FUNCTION_BLOCK FB_MasterArm
VAR
	// arm index, 1 for left arm, 2 for right arm
	m_armIdx: INT;
	
	// grip angle calculator
	m_gripHallSensorIO AT%I* :UDINT;	
	m_gripAngleCalc : FB_GripAngleCalc;
	m_gripAngle :LREAL;
	
	//hand clutch switch IO
	m_handClutchIO AT%I*:UDINT;
	m_handClutchCheck :FB_HandClutchCheck;
	m_handClutchSwitch :BOOL;
	
	// joints
	// NOTICE: all joints are the true active joints, not DH ones!
	m_joints :ARRAY[1..g_mJntNum] OF FB_ArmJoint;
	
	// master gripper roll flip flag, if true, q7 would add pi in FK
	m_gripperRollFlip :BOOL :=False;
	
	// arm cartesian data, defined in each arm origin
	m_curCartPose	:ST_Frame;
	m_curCartTwist: Vec6d;
	m_cmdCartTwist :Vec6d;
	m_cmdCartPose:ST_Frame;
	m_curCartLinkPose :ST_Frame;
	m_curCartLinkTwist :Vec6d;
	
	
	// arm joint data
	m_curMotorPos :Vec7d;
	m_curLinkPos :Vec7d;
	m_curJntPos :Vec7d;
	m_curJntVel :Vec7d;
	m_curLinkVel :Vec7d;
	m_curJntTrq :Vec7d;
	m_rawJntCurrent :Vec7d;
	m_filtJntCurrent :Vec7d;
	m_cmdJntCurrent : Vec7d;
	m_cmdJntTrq :Vec7d;
	m_cmdJntPos :Vec7d;
	m_cmdJntVel :Vec7d;

	
	// arm dynamic data
	m_jntGravity : Vec7d;
	m_jntMassMat : Mat7d;
	m_lambda :Mat6d;
	m_dynaNullspace :Mat7d;
	m_jntFriction :Vec7d;
	m_jntExtTrq :Vec7d;
	
	// arm jacobian 
	m_jaco : Mat67;
	m_linkJaco : Mat67;
	
	// simulated status
	m_simJntPos :Vec7d;
	m_simCartPose : ST_Frame;
	m_simJaco : Mat67;
	
	// joint position controller
	m_jntPIDCtrl :ARRAY[1..g_mJntNum] OF FB_PID;
	
	//inertia compensation---1106
	m_curJntAcc :Vec7d;
	m_curLinkAcc :Vec7d;
	m_jntInertiaTrq:Vec7d;
	m_linkInertiaTrq:Vec7d;	
	
	//Calculate space velocity related variables
	m_linkJacoLast : Mat67; //last link jacobian matrix
	m_spaceAcc:Vec6d; //space acceleration
	m_spaceAccByDiff:Vec6d;
	m_curCartLinkTwistLast :Vec6d;	
	
	//Spatial force related variables
	m_spatialForce:Vec6d;
	m_spatialForceByAccDiff:Vec6d;
	m_jntTorForAcc:Vec7d;
	m_jntTorForAccByDiff:Vec7d;
	
	//Spatial acceleration filter
	m_spatialAccLpf :ARRAY[1..6] OF FB_LowPassFilter;
	m_spatialAccLpf_2 :ARRAY[1..6] OF FB_LowPassFilter;
END_VAR

PROPERTY armIdx : int
GET
armIdx:=m_armIdx;
END_GET
END_PROPERTY

METHOD PROTECTED calcJaco : BOOL
VAR_IN_OUT CONSTANT
	i_jntPos :ARRAY[1..g_mJntNum] OF LREAL;
END_VAR
VAR_IN_OUT
	r_jaco :ARRAY[1..g_cartDofs, 1..g_mJntNum] OF LREAL;
END_VAR
VAR_INPUT
END_VAR

VAR
	q1,q2, q3, q4, q5, q6, q7 :LREAL;
	d1,d4,a3,a4 :LREAL;
	c1,c2,c3,c4,c5,c6,c7 :LREAL;
	s1,s2,s3,s4,s5,s6,s7 :LREAL;
	c23, s23 :LREAL;
	j:INT;
END_VAR
// !Convert active joint position to DH model for kinematic calculation
q1:=i_jntPos[1];  
q2:=i_jntPos[2];  
q3:=i_jntPos[3]-i_jntPos[2];  //q3=q8-q2
q4:=i_jntPos[4]+i_jntPos[3]-i_jntPos[2]-pi/2;//q4DH=q4motor+q8-q2-90;  
q5:=i_jntPos[5];  
q6:=i_jntPos[6];  
q7:=i_jntPos[7];  
d1:=g_d1;
d4:=g_d4;
a3:=g_a3;
a4:=g_a4;
c1:=COS(q1);
c2:=COS(q2);
c3:=COS(q3);
c4:=COS(q4);
c5:=COS(q5);
c6:=COS(q6);
c7:=COS(q7);
s1:=SIN(q1);
s2:=SIN(q2);
s3:=SIN(q3);
s4:=SIN(q4);
s5:=SIN(q5);
s6:=SIN(q6);
s7:=SIN(q7);
c23:=COS(q2+q3);
s23:=SIN(q2+q3);

// jacobian with DH joints
r_jaco[1,1]:=-s1*(c2*(a3 + a4*c3 - d4*s3) - s2*(d4*c3 + a4*s3)) ;
r_jaco[1,2]:=-c1*(s2*(a3 + a4*c3 - d4*s3) + c2*(d4*c3 + a4*s3)) ;
r_jaco[1,3]:=-c1*(d4*c23 + a4*s23) ;
r_jaco[1,4]:=0 ;
r_jaco[1,5]:=0 ;
r_jaco[1,6]:=0 ;
r_jaco[1,7]:=0;
 
r_jaco[2,1]:=c1*(c2*(a3 + a4*c3 - d4*s3) - s2*(d4*c3 + a4*s3)); 
r_jaco[2,2]:=-s1*(s2*(a3 + a4*c3 - d4*s3) + c2*(d4*c3 + a4*s3)); 
r_jaco[2,3]:=-s1*(d4*c23 + a4*s23); 
r_jaco[2,4]:=0; 
r_jaco[2,5]:=0; 
r_jaco[2,6]:=0; 
r_jaco[2,7]:=0;

 
r_jaco[3,1]:=0 ;
r_jaco[3,2]:=- c1*(c1*c2*(a3 + a4*c3 - d4*s3) - c1*s2*(d4*c3 + a4*s3)) - s1*(c2*s1*(a3 + a4*c3 - d4*s3) - s1*s2*(d4*c3 + a4*s3));
r_jaco[3,3]:=- c1*(a4*c23*c1 - d4*s23*c1) - s1*(a4*c23*s1 - d4*s23*s1);
r_jaco[3,4]:=0;
r_jaco[3,5]:=0;
r_jaco[3,6]:=0 ;
r_jaco[3,7]:=0 ;

r_jaco[4,1]:=0 ;
r_jaco[4,2]:=-s1 ;
r_jaco[4,3]:=-s1 ;
r_jaco[4,4]:=-s23*c1 ;
r_jaco[4,5]:=c23*c1*s4 - c4*s1 ;
r_jaco[4,6]:=- s5*(s1*s4 + c23*c1*c4) - s23*c1*c5 ;
r_jaco[4,7]:=s6*(c5*(s1*s4 + c4*(c1*c2*c3 - c1*s2*s3)) - s5*(c1*c2*s3 + c1*c3*s2)) - c6*(c4*s1 - s4*(c1*c2*c3 - c1*s2*s3));
 
r_jaco[5,1]:=0; 
r_jaco[5,2]:=c1; 
r_jaco[5,3]:=c1; 
r_jaco[5,4]:=-s23*s1; 
r_jaco[5,5]:=c1*c4 + c23*s1*s4; 
r_jaco[5,6]:=s5*(c1*s4 - c23*c4*s1) - s23*c5*s1; 
r_jaco[5,7]:=c6*(c1*c4 - s4*(s1*s2*s3 - c2*c3*s1)) - s6*(c5*(c1*s4 + c4*(s1*s2*s3 - c2*c3*s1)) + s5*(c2*s1*s3 + c3*s1*s2));

r_jaco[6,1]:=1 ;
r_jaco[6,2]:=0 ;
r_jaco[6,3]:=0 ;
r_jaco[6,4]:=-c23 ;
r_jaco[6,5]:=-s23*s4 ;
r_jaco[6,6]:=s23*c4*s5 - c23*c5 ;
r_jaco[6,7]:=- s6*(c23*s5 + s23*c4*c5) - s23*c6*s4;

// jacobian with active joints
// jaco_DH*qdot_DH = jaco_DH * (A * qdot)= jaco * qdot
// A =[ 1  0 0 0 0 0 0
//		0  1 0 0 0 0 0
//		0 -1 1 0 0 0 0
//		0 -1 1 1 0 0 0
//		0 0  0 0 1 0 0
//      0 0  0 0 0 1 0
// 		0 0  0 0 0 0 1]
 FOR j:=1 TO 6 DO 
	 r_jaco[j,2]:=r_jaco[j,2]-r_jaco[j,3]-r_jaco[j,4];
	 r_jaco[j,3]:=r_jaco[j,3]+r_jaco[j,4];
 END_FOR
END_METHOD

PROPERTY cmdCartPose : REFERENCE TO ST_Frame
GET
cmdCartPose REF= m_cmdCartPose;
END_GET
END_PROPERTY

PROPERTY cmdCartTwist : REFERENCE to Vec6d
GET
cmdCartTwist REF= m_cmdCartTwist;
END_GET
END_PROPERTY

PROPERTY cmdJntCurrent :REFERENCE to Vec7d
GET
cmdJntCurrent REF= m_cmdJntCurrent;
END_GET
END_PROPERTY

PROPERTY cmdJntPos : REFERENCE TO Vec7d
GET
cmdJntPos REF= m_cmdJntPos;
END_GET
END_PROPERTY

PROPERTY cmdJntTrq :REFERENCE TO Vec7d
GET
cmdJntTrq REF= m_cmdJntTrq;
END_GET
END_PROPERTY

PROPERTY cmdJntVel : REFERENCE TO Vec7d
GET
cmdJntVel REF= m_cmdJntVel;
END_GET
END_PROPERTY

PROPERTY curCartPose :REFERENCE to ST_Frame
GET
curCartPose REF=m_curCartPose;
END_GET
END_PROPERTY

PROPERTY curCartTwist :REFERENCE TO Vec6d
GET
curCartTwist REF=m_curCartTwist;
END_GET
END_PROPERTY

PROPERTY curJntInertiaTrq :REFERENCE TO Vec7d
GET

//cmdJntPos REF= m_cmdJntPos;---inertia compensation---1106
IF (gvl.m_InertiaSelect[m_armIdx]=1) THEN
	curJntInertiaTrq REF=m_jntInertiaTrq;
	
ELSIF(gvl.m_InertiaSelect[m_armIdx]=2) THEN
	curJntInertiaTrq REF=m_linkInertiaTrq;
	
ELSIF(gvl.m_InertiaSelect[m_armIdx]=3) THEN
	curJntInertiaTrq REF=m_jntTorForAcc;
	
ELSIF(gvl.m_InertiaSelect[m_armIdx]=4) THEN
	curJntInertiaTrq REF=m_jntTorForAccByDiff;
END_IF
END_GET
SET
END_SET
END_PROPERTY

PROPERTY curJntPos :REFERENCE TO Vec7d
GET
curJntPos REF=m_curJntPos;
END_GET
END_PROPERTY

PROPERTY curJntTrq :REFERENCE TO Vec7d
GET
curJntTrq REF=m_curJntTrq;
END_GET
END_PROPERTY

PROPERTY curJntVel :REFERENCE TO Vec7d
GET
curJntVel REF=m_curJntVel;
END_GET
END_PROPERTY

PROPERTY curLinkPos :REFERENCE TO  Vec7d
GET
curLinkPos REF=m_curLinkPos;
END_GET
END_PROPERTY

PROPERTY curMotorPos :REFERENCE TO Vec7d
GET
curMotorPos REF=m_curMotorPos;
END_GET
END_PROPERTY

PROPERTY PUBLIC dynaNullspace : REFERENCE TO Mat7d
GET
dynaNullspace REF= m_dynaNullspace;
END_GET
END_PROPERTY

METHOD PROTECTED enable : BOOL
VAR_IN_OUT CONSTANT
	i_jntIdx :Vec7i;
END_VAR
VAR
	i :INT ;
END_VAR
FOR i:=1 TO g_mJntNum DO
	IF 1= i_jntIdx[i] THEN
		m_joints[i].enable();
	ELSE
		m_joints[i].disable();
	END_IF
END_FOR
END_METHOD

PROPERTY filtJntCurrent :REFERENCE to Vec7d
GET
filtJntCurrent ref= m_filtJntCurrent;
END_GET
END_PROPERTY

METHOD PUBLIC flipGripper : BOOL
VAR_INPUT
	i_flipFlag :BOOL;
END_VAR
m_gripperRollFlip := i_flipFlag;
END_METHOD

// from active joint position to cartesian pose in arm origin
METHOD PROTECTED forwardKinematic : BOOL
VAR_IN_OUT CONSTANT
	i_jntPos :ARRAY[1..g_mJntNum] OF LREAL;
END_VAR
VAR_IN_OUT
	r_cartPose :ST_Frame;
END_VAR
VAR
	q1,q2, q3, q4, q5, q6, q7 :LREAL;
	d1,d4,a3,a4 :LREAL;
	c1,c2,c3,c4,c5,c6,c7 :LREAL;
	s1,s2,s3,s4,s5,s6,s7 :LREAL;
	c23, s23 :LREAL;
END_VAR
// !Convert active joint position to DH model for kinematic calculation
q1:=i_jntPos[1];  
q2:=i_jntPos[2];  
q3:=i_jntPos[3]-i_jntPos[2];  //q3=q8-q2
q4:=jnt4MotorToLink(i_jntPos[2],i_jntPos[3], i_jntPos[4]);//q4DH=q4motor+q8-q2-90;  
q5:=i_jntPos[5];  
q6:=i_jntPos[6];  
q7:=i_jntPos[7];  

// master roll flip handle
IF m_gripperRollFlip THEN
	q7 := q7+PI;
END_IF

d1:=g_d1;
d4:=g_d4;
a3:=g_a3;
a4:=g_a4;
c1:=COS(q1);
c2:=COS(q2);
c3:=COS(q3);
c4:=COS(q4);
c5:=COS(q5);
c6:=COS(q6);
c7:=COS(q7);
s1:=SIN(q1);
s2:=SIN(q2);
s3:=SIN(q3);
s4:=SIN(q4);
s5:=SIN(q5);
s6:=SIN(q6);
s7:=SIN(q7);
c23:=COS(q2+q3);
s23:=SIN(q2+q3);

// cartesian pose frame
r_cartPose.m_pos[1]:=c1*(a4*c23 - d4*s23 + a3*c2); 
r_cartPose.m_pos[2]:=s1*(a4*c23 - d4*s23 + a3*c2);
r_cartPose.m_pos[3]:=d1 - d4*c23 - a4*s23 - a3*s2;  
r_cartPose.m_rot[1,1]:=c7*(s6*(c4*s1 - s4*(c1*c2*c3 - c1*s2*s3)) + c6*(c5*(s1*s4 + c4*(c1*c2*c3 - c1*s2*s3)) - s5*(c1*c2*s3 + c1*c3*s2))) - s7*(s5*(s1*s4 + c4*(c1*c2*c3 - c1*s2*s3)) + c5*(c1*c2*s3 + c1*c3*s2));
r_cartPose.m_rot[2,1]:=s7*(s5*(c1*s4 + c4*(s1*s2*s3 - c2*c3*s1)) - c5*(c2*s1*s3 + c3*s1*s2)) - c7*(s6*(c1*c4 - s4*(s1*s2*s3 - c2*c3*s1)) + c6*(c5*(c1*s4 + c4*(s1*s2*s3 - c2*c3*s1)) + s5*(c2*s1*s3 + c3*s1*s2)));
r_cartPose.m_rot[3,1]:=- s7*(c23*c5 - s23*c4*s5) - c7*(c23*c6*s5 - s23*s4*s6 + s23*c4*c5*c6); 
r_cartPose.m_rot[1,2]:=- s7*(s6*(c4*s1 - s4*(c1*c2*c3 - c1*s2*s3)) + c6*(c5*(s1*s4 + c4*(c1*c2*c3 - c1*s2*s3)) - s5*(c1*c2*s3 + c1*c3*s2))) - c7*(s5*(s1*s4 + c4*(c1*c2*c3 - c1*s2*s3)) + c5*(c1*c2*s3 + c1*c3*s2)); 
r_cartPose.m_rot[2,2]:=s7*(s6*(c1*c4 - s4*(s1*s2*s3 - c2*c3*s1)) + c6*(c5*(c1*s4 + c4*(s1*s2*s3 - c2*c3*s1)) + s5*(c2*s1*s3 + c3*s1*s2))) + c7*(s5*(c1*s4 + c4*(s1*s2*s3 - c2*c3*s1)) - c5*(c2*s1*s3 + c3*s1*s2)); 
r_cartPose.m_rot[3,2]:=s7*(c23*c6*s5 - s23*s4*s6 + s23*c4*c5*c6) - c7*(c23*c5 - s23*c4*s5); 
r_cartPose.m_rot[1,3]:=s6*(c5*(s1*s4 + c4*(c1*c2*c3 - c1*s2*s3)) - s5*(c1*c2*s3 + c1*c3*s2)) - c6*(c4*s1 - s4*(c1*c2*c3 - c1*s2*s3)); 
r_cartPose.m_rot[2,3]:=c6*(c1*c4 - s4*(s1*s2*s3 - c2*c3*s1)) - s6*(c5*(c1*s4 + c4*(s1*s2*s3 - c2*c3*s1)) + s5*(c2*s1*s3 + c3*s1*s2));
r_cartPose.m_rot[3,3]:=- s6*(c23*s5 + s23*c4*c5) - s23*c6*s4;
END_METHOD

PROPERTY gripAngle : LREAL
GET
gripAngle:=m_gripAngle;
END_GET
END_PROPERTY

PROPERTY gripperRollFlip : BOOL
GET
gripperRollFlip := m_gripperRollFlip;
END_GET
END_PROPERTY

PROPERTY handClutchSwitch : BOOL
GET
handClutchSwitch :=m_handClutchSwitch;
END_GET
END_PROPERTY

METHOD PUBLIC init : BOOL
VAR_INPUT
	i_armIdx:INT;
END_VAR
VAR 
	i :INT ;
	currentRatioMotor2Jnt: LREAL;
END_VAR
// arm statues init
m_armIdx:=i_armIdx;
m_gripAngle:=0;
m_gripAngleCalc.init(m_armIdx);

// joint init
FOR i:=1 TO g_mJntNum DO
	m_joints[i].init(m_armIdx, i,g_armCtrlCycleTime);
END_FOR

// init joint encoder and position calculation
initJntPos();

// joint controller init
FOR i:=1 TO g_mJntNum DO 
	currentRatioMotor2Jnt:=GVL_ArmJointParameters.g_motorTrqConst[i]*GVL_ArmJointParameters.g_motorReduction[i]/1000;
	m_jntPIDCtrl[i].init(g_armCtrlCycleTime,g_posKp[i],g_posKd[i],g_posKi[i],
		g_posKiLimit[i]* currentRatioMotor2Jnt,	g_posCtrlLimit[i]*currentRatioMotor2Jnt);
END_FOR

//spatial acceleration init---inertia compensation---1106
FOR i:=1 TO 6 DO 
	m_spatialAccLpf[i].init(1, g_curJntVelLpfCutoffFreq*0.2, g_armCtrlFreq/gvl.g_accCalCycle);
	m_spatialAccLpf_2[i].init(1, g_curJntVelLpfCutoffFreq*0.2, g_armCtrlFreq/gvl.g_accCalCycle);
END_FOR
END_METHOD

METHOD public initJntPos : BOOL
VAR_INPUT
END_VAR
VAR
	i:INT ;
	initLinkPos:LREAL;
END_VAR
// joint init
FOR i:=1 TO g_mJntNum DO
	m_joints[i].initJntPos();
END_FOR

// link position of joint4 is influenced by joint2 and joint3, need to handle seperately
initLinkPos:=jnt4LinkToMotor(m_joints[2].initLinkPos,m_joints[3].initLinkPos, m_joints[4].initLinkPos);
m_joints[4].initJntPosReset(initLinkPos);

// update arm status after joint position is re-init
updateStatus();
END_METHOD

// from cartesian pose in arm origin to active joint position
METHOD PROTECTED inverseKinematic : BOOL
VAR_INPUT
	q4:LREAL;
	solution_ID:INT;
END_VAR
VAR_IN_OUT CONSTANT
	i_curCartPose :ST_Frame;
END_VAR
VAR_IN_OUT
	r_jntPos :ARRAY[1..g_mJntNum] OF LREAL;
END_VAR
VAR
	a3,a4,d1,d4:LREAL;
	px,py,pz:lreal;
	nx,ny,nz:lreal;
	ox,oy,oz:lreal;
	ax,ay,az:lreal;

	q1,q2,q3,q5,q6,q7:LREAL;
	
	q11,q12:LREAL;
	k1,A,B,C,fi,R0,q21,q22:lreal;
	ins1,ins2:lreal;
	
	A11,A12,A21,A22,C1,C2:lreal;
	SIN23,COS23,q23:lreal;
	
	T_74_left_23,q61,q62:lreal;
	T_74_left_13,T_74_left_33:lreal;
	T_74_left_21,T_74_left_22:LREAL;	
	
	succeed_1,succeed_2,succeed:BOOL;
END_VAR


//***********************单臂逆向运动学**************************//
d1:=g_d1;
d4:=g_d4;
a3:=g_a3;
a4:=g_a4;

nx:=i_curCartPose.m_rot[1,1];  ny:=i_curCartPose.m_rot[2,1];  nz:=i_curCartPose.m_rot[3,1];
ox:=i_curCartPose.m_rot[1,2]; oy:=i_curCartPose.m_rot[2,2];  oz:=i_curCartPose.m_rot[3,2];
ax:=i_curCartPose.m_rot[1,3];  ay:=i_curCartPose.m_rot[2,3];  az:=i_curCartPose.m_rot[3,3];
px:=i_curCartPose.m_pos[1]; py:=i_curCartPose.m_pos[2]; pz:=i_curCartPose.m_pos[3];


//求解q1
q11:=atan2(y:= py, x:= px);
q12:=-q11;
IF (Solution_ID<=4) THEN
	q1:=q11;
ELSE
	q1:=q12;
END_IF



//求解q2
k1:=px*COS(q1) + py*SIN(q1);
A:=2*a3*pz - 2*a3*d1;
B:=2*a3*k1;
C:=a3*a3 - a4*a4 + d1*d1 - 2*d1*pz - d4*d4 + k1*k1 + pz*pz;
fi:=atan2(y:= B, x:= A);

R0:=SQRT(A*A+B*B);

//*************程序保护性处理，避免软件崩溃***************//
IF ABS(C/R0)>1 THEN
	succeed_1:=FALSE;
	succeed:=FALSE;
	RETURN;
ELSE
	succeed_1:=TRUE;
END_IF

ins1:=atan2(y:= C/R0, x:= SQRT(1-(C/R0)*(C/R0)));
q21:=fi-ins1;
ins2:=atan2(y:= C/R0, x:= -SQRT(1-(C/R0)*(C/R0)));
q22:=fi-ins2;

IF (Solution_ID=1) OR (Solution_ID=2) OR (Solution_ID=5) OR (Solution_ID=6) THEN
	q2:=q21;
ELSE
	q2:=q22;
END_IF




//求解q3
A11:=- d4;
A12:=a4;
A21:=- a4;
A22:=-d4;
C1:=k1- a3*COS(q2);
C2:=pz - d1 + a3*SIN(q2);
sin23:=(C1*A22-C2*A12)/(A11*A22-A21*A12);
cos23:=(C2*A11-C1*A21)/(A11*A22-A21*A12);
q23:=atan2(y:= sin23, x:= cos23);
q3:=q23-q2;




//求解q6
T_74_left_23:=ax*(COS(q4)*SIN(q1) - COS(q1)*COS(q2)*COS(q3)*SIN(q4) + COS(q1)*SIN(q2)*SIN(q3)*SIN(q4)) - ay*(COS(q1)*COS(q4) + COS(q2)*COS(q3)*SIN(q1)*SIN(q4) - SIN(q1)*SIN(q2)*SIN(q3)*SIN(q4)) + az*SIN(q2 + q3)*SIN(q4);

//*************程序保护性处理，避免软件崩溃***************//
IF ABS(T_74_left_23>1) THEN
	succeed_2:=FALSE;
	succeed:=FALSE;
	RETURN;
ELSE
	succeed_2:=TRUE;
END_IF

q61:=ACOS(-T_74_left_23);
q62:=-ACOS(-T_74_left_23);
IF (Solution_ID=1) OR (Solution_ID=3) OR (Solution_ID=5) OR (Solution_ID=7) THEN
	q6:=q61;
ELSE
	q6:=q62;
END_IF


//求解q5
T_74_left_13:=ax*(SIN(q1)*SIN(q4) + COS(q1)*COS(q2)*COS(q3)*COS(q4) - COS(q1)*COS(q4)*SIN(q2)*SIN(q3)) - ay*(COS(q1)*SIN(q4) - COS(q2)*COS(q3)*COS(q4)*SIN(q1) + COS(q4)*SIN(q1)*SIN(q2)*SIN(q3)) - az*SIN(q2 + q3)*COS(q4);
T_74_left_33:=- az*COS(q2 + q3) - ax*SIN(q2 + q3)*COS(q1) - ay*SIN(q2 + q3)*SIN(q1);
q5:=atan2(y:= T_74_left_33*SIN(q6), x:= T_74_left_13*SIN(q6));


//求解q7
T_74_left_21:=nx*(COS(q4)*SIN(q1) - COS(q1)*COS(q2)*COS(q3)*SIN(q4) + COS(q1)*SIN(q2)*SIN(q3)*SIN(q4)) - ny*(COS(q1)*COS(q4) + COS(q2)*COS(q3)*SIN(q1)*SIN(q4) - SIN(q1)*SIN(q2)*SIN(q3)*SIN(q4)) + nz*SIN(q2 + q3)*SIN(q4);
T_74_left_22:=ox*(COS(q4)*SIN(q1) - COS(q1)*COS(q2)*COS(q3)*SIN(q4) + COS(q1)*SIN(q2)*SIN(q3)*SIN(q4)) - oy*(COS(q1)*COS(q4) + COS(q2)*COS(q3)*SIN(q1)*SIN(q4) - SIN(q1)*SIN(q2)*SIN(q3)*SIN(q4)) + oz*SIN(q2 + q3)*SIN(q4);
q7:=atan2(y:= -T_74_left_22*SIN(q6), x:= T_74_left_21*SIN(q6));


//! convert DH joint postion to active joint position
r_jntPos[1]:=q1;
r_jntPos[2]:=q2;
r_jntPos[3]:=q3+q2; // q8 = q3+q2
r_jntPos[4]:=q4+q2-r_jntPos[3]+pi/2;//q4DH=q4motor+q8-q2-90;  
r_jntPos[5]:=q5;
r_jntPos[6]:=q6;
r_jntPos[7]:=q7;

succeed:=TRUE;
inverseKinematic:=succeed;
END_METHOD

METHOD PUBLIC isEnabled : BOOL
VAR_IN_OUT CONSTANT
	i_jntIdx :Vec7i;
END_VAR
VAR
	i :INT ;
END_VAR
isEnabled := TRUE;
FOR i:=1 TO g_mJntNum DO
	IF 1= i_jntIdx[i] THEN
		isEnabled :=  (m_joints[i].isEnabled() AND isEnabled);
	END_IF
END_FOR
END_METHOD

PROPERTY jaco :REFERENCE to Mat67
GET
jaco ref= m_jaco;
END_GET
END_PROPERTY

//convert joint4 position from link side to motor side
METHOD PUBLIC jnt4LinkToMotor : LREAL
VAR_INPUT
	i_q2 :LREAL;
	i_q3:LREAL;
	i_q4Link :LREAL;
END_VAR
jnt4LinkToMotor:=i_q4Link-i_q3+i_q2+pi/2;//q4motor=q4DH-q8+q2+90;
END_METHOD

//convert joint4 position from motor side to link side
METHOD public jnt4MotorToLink : LREAL
VAR_INPUT
	i_q2 :LREAL;
	i_q3:LREAL;
	i_q4Motor :LREAL;
END_VAR
jnt4MotorToLink:=i_q4Motor+i_q3-i_q2-pi/2;//q4DH=q4motor+q8-q2-90;
END_METHOD

PROPERTY jntExtTrq :REFERENCE TO Vec7d
GET
jntExtTrq REF= m_jntExtTrq;
END_GET
END_PROPERTY

PROPERTY jntFriction :REFERENCE TO Vec7d
GET
jntFriction REF= m_jntFriction;
END_GET
END_PROPERTY

PROPERTY jntGravity :REFERENCE to Vec7d
GET
jntGravity ref=m_jntGravity;
END_GET
END_PROPERTY

PROPERTY PUBLIC massMat :REFERENCE to Mat7d
GET
massMat ref=m_jntMassMat;
END_GET
END_PROPERTY

PROPERTY rawJntCurrent :REFERENCE to Vec7d
GET
rawJntCurrent ref=m_rawJntCurrent;
END_GET
END_PROPERTY

PROPERTY simCartPose :REFERENCE to ST_Frame
GET
simCartPose REF=m_simCartPose;
END_GET
END_PROPERTY

PROPERTY simJaco :REFERENCE TO mat67
GET
simJaco REF=m_simJaco;
END_GET
END_PROPERTY

// update joints control command
METHOD PUBLIC updateCmds : BOOL
VAR_IN_OUT CONSTANT
	i_armCtrlCmd : ST_ArmCtrlCmds;
END_VAR
VAR
	i:INT;
END_VAR
m_cmdJntTrq:=i_armCtrlCmd.m_cmdJntTrq;
m_cmdJntPos :=i_armCtrlCmd.m_cmdJntPos;
m_cmdJntVel :=i_armCtrlCmd.m_cmdJntVel;
m_cmdCartTwist := i_armCtrlCmd.m_cmdCartTwist;
m_cmdCartPose :=i_armCtrlCmd.m_cmdCartPose;
m_simJntPos:=i_armCtrlCmd.m_cmdJntPos;

// update simulated master arm
updateSimStatus();

// enable/disable joints
enable(i_armCtrlCmd.m_jntEnableFlag);

// position/torque control
FOR i:=1 TO g_mJntNum DO 
	IF i_armCtrlCmd.m_jntOPMode[i]=DriverOPMode_PosTrq THEN
		// position controller and gravity feedforward
		m_cmdJntTrq[i]:=m_jntPIDCtrl[i].run(i_armCtrlCmd.m_cmdJntPos[i],m_curJntPos[i],i_armCtrlCmd.m_cmdJntVel[i],m_curJntVel[i]);
		m_cmdJntTrq[i]:=m_cmdJntTrq[i]+m_jntGravity[i];
		m_joints[i].updateCmds(DriverOPMode_Trq,i_armCtrlCmd.m_cmdJntPos[i],m_cmdJntTrq[i]);
	ELSIF i_armCtrlCmd.m_jntOPMode[i]=DriverOPMode_Trq THEN
		// gravity feedforward
		m_jntPIDCtrl[i].reset();
		m_cmdJntTrq[i]:=m_cmdJntTrq[i]+m_jntGravity[i];
		m_joints[i].updateCmds(DriverOPMode_Trq,i_armCtrlCmd.m_cmdJntPos[i],m_cmdJntTrq[i]);
	ELSE
		m_jntPIDCtrl[i].reset();
		m_cmdJntTrq[i]:=0;
		m_joints[i].updateCmds(DriverOPMode_Pos,i_armCtrlCmd.m_cmdJntPos[i],m_cmdJntTrq[i]);
	END_IF
	
END_FOR
END_METHOD

METHOD PUBLIC updateDyna : BOOL
VAR_IN_out constant
	masterDynaData : ST_MasterDynaData;
END_VAR
m_jntMassMat:=masterDynaData.m_massMat[m_armIdx];
m_lambda:=masterDynaData.m_lambda[m_armIdx];
m_dynaNullspace:=masterDynaData.m_dynaNullspace[m_armIdx];
m_jntGravity:=masterDynaData.m_gravity[m_armIdx];
m_jntFriction:=masterDynaData.m_friction[m_armIdx];
m_jntExtTrq := masterDynaData.m_jntExtTrq[m_armIdx];
END_METHOD

METHOD PUBLIC updateSimStatus : BOOL
VAR_INPUT
END_VAR
// simulated cartesion pose 
forwardKinematic(m_simJntPos,m_simCartPose);

// simulated jacobian
calcJaco(m_simJntPos,m_simJaco);
END_METHOD

// update arm status, including kinematic and dynamic
METHOD PUBLIC updateStatus : BOOL
VAR_INPUT
END_VAR
VAR 
	i,j:INT;
	tmpMat67 : Mat67;
	JacoDot:Mat67;
	JacoT:Mat76;
	spaceAccPart1,spaceAccPart2:Vec6d;
	curCartLinkTwistDiff :Vec6d;
	factor:LREAL;
END_VAR
// grip angle
m_gripAngle :=m_gripAngleCalc.run(m_gripHallSensorIO);

// check hand clutch
m_handClutchSwitch :=  m_handClutchCheck.run(m_handClutchIO);

// update joint data
FOR i:=1 TO g_mJntNum DO
	m_joints[i].updateStatus();
END_FOR

// get joint data
FOR i:=1 TO g_mJntNum DO
	m_curMotorPos[i]:=m_joints[i].motorPos;
	m_curLinkPos[i]:=m_joints[i].linkPos;
	m_curJntPos[i]:=m_joints[i].jntPos;
	m_curJntVel[i]:=m_joints[i].jntVel;
	m_curLinkVel[i] := m_joints[i].m_curLinkVel;
	
	m_curJntAcc[i]:=m_joints[i].m_curJntAcc; //inertia compensation---1106
	m_curLinkAcc[i]:=m_joints[i].m_curLinkAcc;
	
	m_curJntTrq[i]:=m_joints[i].jntTrq;
	m_rawJntCurrent[i]:=m_joints[i].rawCurrent;
	m_filtJntCurrent[i]:=m_joints[i].filtCurrent;
	m_cmdJntCurrent[i]:=m_joints[i].cmdCurrent;
END_FOR 
m_curLinkPos[4]:=jnt4LinkToMotor(m_curLinkPos[2],m_curLinkPos[3], m_curLinkPos[4]);// q4motor=q4DH-q8+q2+90; 
m_curLinkVel[4]:= m_curLinkVel[4] - m_curLinkVel[3] + m_curLinkVel[2]; 

//inertia compensation---1106
m_curLinkAcc[4]:= m_curLinkAcc[4] - m_curLinkAcc[3] + m_curLinkAcc[2];

// cartesion pose
forwardKinematic(m_curJntPos,m_curCartPose);
forwardKinematic(m_curLinkPos,m_curCartLinkPose);

// jacobian
calcJaco(m_curJntPos,m_jaco);
calcJaco(m_curLinkPos,m_linkJaco);

// cartesian twist
matMultiVec(m_jaco,m_curJntVel,m_curCartTwist);
matMultiVec(m_linkJaco,m_curLinkVel,m_curCartLinkTwist);


//joint inertia torque--- //inertia compensation---1106
matMultiVec(m_jntMassMat,m_curJntAcc,m_jntInertiaTrq);
//m_curLinkAcc[4]:=0;
matMultiVec(m_jntMassMat,m_curLinkAcc,m_linkInertiaTrq);


//Calculate inertial forces in the operating space
IF (m_joints[1].m_accCycle=0) THEN
	//taking the derivative of the Jacobian matrix
	matSub(m_linkJaco,m_linkJacoLast,tmpMat67);
	factor:=1.0/(gvl.g_accCalCycle*g_armCtrlCycleTime);
	matMultiNum(tmpMat67,factor,JacoDot);
	m_linkJacoLast:=m_linkJaco;
	
	//Calculate spatial acceleration and filter it
	matMultiVec(JacoDot,m_curLinkVel,spaceAccPart1);
	matMultiVec(m_linkJaco,m_curLinkAcc,spaceAccPart2);
	vecAdd(spaceAccPart1,spaceAccPart2,m_spaceAcc);
	FOR i:=1 TO 6 BY 1 DO
		//m_spaceAcc[i]:=m_spatialAccLpf[i].run(m_spaceAcc[i]);
	END_FOR
	
	//Calculate the inertial force of the operating space
	matMultiVec(m_lambda,m_spaceAcc,m_spatialForce);
	matTranspose(m_linkJaco,JacoT);
	matMultiVec(JacoT,m_spatialForce,m_jntTorForAcc);		
	
	//taking the derivative of spatial velocity
	vecSub(m_curCartLinkTwist,m_curCartLinkTwistLast,curCartLinkTwistDiff);
	vecMultiNum(curCartLinkTwistDiff,1.0/(gvl.g_accCalCycle*g_armCtrlCycleTime),m_spaceAccByDiff);
	m_curCartLinkTwistLast:=m_curCartLinkTwist;
	FOR i:=1 TO 6 BY 1 DO
		m_spaceAccByDiff[i]:=m_spatialAccLpf_2[i].run(m_spaceAccByDiff[i]);
	END_FOR
	
	//Calculate the inertial force of the operating space and convert it into joint torque
	matMultiVec(m_lambda,m_spaceAccByDiff,m_spatialForceByAccDiff);
	matMultiVec(JacoT,m_spatialForceByAccDiff,m_jntTorForAccByDiff);
END_IF


//Inertia force scaling factor
FOR i:=1 TO g_mJntNum DO
	gvl.g_jntVelFactor[m_armIdx,i]:=LIMIT(0,ABS(m_curLinkVel[i]/(gvl.g_jntVelLimit[m_armIdx,i]*gvl.g_jntVelLimitScaler[m_armIdx])),1);
	gvl.g_jntAccFactor[m_armIdx,i]:=LIMIT(0,ABS(m_curLinkAcc[i]/gvl.g_jntAccLimit[m_armIdx,i]*gvl.g_jntAccLimitScaler[m_armIdx]),1);
END_FOR


(*
//Program debugging related variables
gvl.m_curJntPos[m_armIdx]:=m_curJntPos;
gvl.m_curJntVel[m_armIdx]:=m_curJntVel;
gvl.m_curJntAcc[m_armIdx]:=m_curJntAcc;

gvl.m_jntInertiaTrq[m_armIdx]:=m_jntInertiaTrq;
gvl.m_linkInertiaTrq[m_armIdx]:=m_linkInertiaTrq;

gvl.m_curLinkPos[m_armIdx]:=m_curLinkPos;
gvl.m_curLinkVel[m_armIdx]:=m_curLinkVel;
gvl.m_curLinkAcc[m_armIdx]:=m_curLinkAcc;

gvl.m_spaceAcc[m_armIdx]:=m_spaceAcc;
gvl.m_spaceAccByDiff[m_armIdx]:=m_spaceAccByDiff;
gvl.m_jntAccTrq[m_armIdx]:=m_jntTorForAcc;
gvl.m_jntAccTrqByDiff[m_armIdx]:=m_jntTorForAccByDiff;
*)
END_METHOD

END_FUNCTION_BLOCK

(* stored: Version 1.1.0.1, ProductVersion 3.1.4024.11
   POU FB_MasterArm: Id {623926f8-06e2-46b6-bb1f-baa6bc16e9cb}, SpecialFunc None
   Folder property: Id {4aa1799c-1556-4bc1-a713-06f14faa00f1}
   Property armIdx: Id {1bcadfc3-0a4f-4bee-a1a7-b6d4d3a1eb58}
   Get Get: Id {198387ec-2e24-42e6-b0c2-2f769705d46f}
   Method calcJaco: Id {1172e5e4-b7f2-4690-a821-6304414cea84}
   Property cmdCartPose: Id {72bf034f-e694-478b-8fc6-77f6ebb37ccd}
   Get Get: Id {cf508e47-c40b-4af1-9748-e64ccbaeea52}
   Property cmdCartTwist: Id {db564f7b-db8f-4a3a-ba4b-526788bb30bd}
   Get Get: Id {8a565392-e659-4e2f-8d16-f053ffd74289}
   Property cmdJntCurrent: Id {cbd7aa84-e545-47b8-bdc5-960aa8409c91}
   Get Get: Id {12be56c2-8b79-47d6-b1f2-86b8e0a5f91a}
   Property cmdJntPos: Id {fe3eaf75-296c-46e0-a9c6-f78064c649e8}
   Get Get: Id {21440cc7-9bce-4ec3-adb3-863b046ec9da}
   Property cmdJntTrq: Id {a8b8f509-6313-4dea-add6-0d9f63644d17}
   Get Get: Id {69ae4f04-ab57-4161-852a-de73ff986ad6}
   Property cmdJntVel: Id {8b50ea35-c0ee-4521-ab63-6cd2fbfd419a}
   Get Get: Id {32d77105-7aae-4d69-88ee-4b488832fd1d}
   Property curCartPose: Id {d18be23c-99e5-435e-8688-90e0fb3be9ca}
   Get Get: Id {013b03f6-adb7-4855-b0fe-353f77f67094}
   Property curCartTwist: Id {e4b7010c-887c-41fa-8766-1a9192e9d06a}
   Get Get: Id {b7c89bf7-90fc-4841-be25-e467b1918b68}
   Property curJntInertiaTrq: Id {dc8c6e14-984b-4636-a402-bd51ab028349}
   Get Get: Id {55902a2e-1107-48a4-a950-7ec7d27c7ecd}
   Set Set: Id {4981c8fc-789b-4ed8-b227-6b20cd5233ab}
   Property curJntPos: Id {d72c054a-bae9-44cb-97ff-fe7c76c53cb8}
   Get Get: Id {332d5297-fb56-44bd-a751-714464e0813c}
   Property curJntTrq: Id {8c78ba58-302c-4844-9d36-e487700a0e19}
   Get Get: Id {1767bffb-cddd-4133-ad6f-5125f86340af}
   Property curJntVel: Id {904c68d5-30c9-4ed3-b3c5-6bcd345bcd5a}
   Get Get: Id {0a508621-c577-4d50-8cc3-bd8133f79f72}
   Property curLinkPos: Id {3725bf51-2c50-4574-b2a7-e2af9fd4da29}
   Get Get: Id {cff7c92f-5276-4a58-b7ca-f6248868b409}
   Property curMotorPos: Id {ad9d9e24-10f4-4dc4-b0d2-86517dead53b}
   Get Get: Id {bc557e46-3cdd-47ba-9e7f-cf7525f3969d}
   Property dynaNullspace: Id {872e2eb4-66b0-4b49-98a3-75080f1189e3}
   Get Get: Id {8a06f4b9-0c57-44d4-b602-0075d0a644d1}
   Method enable: Id {596f2892-08b6-4851-84d5-1537c558264e}
   Property filtJntCurrent: Id {1f5e4c97-ef8c-417a-90ec-656c048c0e4f}
   Get Get: Id {34ea0c3d-b0bc-4adb-bbb3-f4ab6640a7ff}
   Method flipGripper: Id {b34dfa37-adbc-4e99-a96a-e20f87ddba4a}
   Method forwardKinematic: Id {182b544f-f7c4-475e-8af7-8c07aa230234}
   Property gripAngle: Id {5187a911-df75-4b56-8b45-38142d9b24de}
   Get Get: Id {871729fd-1ba1-4906-aec3-7d572491feb2}
   Property gripperRollFlip: Id {93c1f56a-60e7-470f-8b01-d27018c6d468}
   Get Get: Id {9fa59e73-352b-4612-8aea-47cc6b1973bb}
   Property handClutchSwitch: Id {0795f1a7-d600-4b6e-a827-c75cf14d164e}
   Get Get: Id {52f21347-ac12-4dc6-990c-bcc0a2a6e983}
   Method init: Id {d7bcc040-c32e-4455-ab43-70de0dc2919e}
   Method initJntPos: Id {56ee4071-fcb1-4318-b1b9-837ea21e1627}
   Method inverseKinematic: Id {a2d4ef4e-dcb4-4918-aceb-3d3fb8d74093}
   Method isEnabled: Id {00a67cf8-62b1-4004-a2ca-9469bb0f3cab}
   Property jaco: Id {2c2ce445-b511-4254-9c8e-e5667e1b6bdb}
   Get Get: Id {27a6e900-c6e6-40c0-aa03-4dc0d1214554}
   Method jnt4LinkToMotor: Id {3d664502-a5ca-4a18-947e-2de6df49b268}
   Method jnt4MotorToLink: Id {73c2344c-abd6-47df-a57c-56c9686be51c}
   Property jntExtTrq: Id {626626ac-4a19-4244-8c4e-4b8e5d00c8e6}
   Get Get: Id {a09a5e22-8056-494a-9352-77be189f5fc1}
   Property jntFriction: Id {adee17cd-b04f-47e3-9783-a1860653d53a}
   Get Get: Id {ed7d4727-a7d8-4feb-9606-8aa7b1aafe25}
   Property jntGravity: Id {72dbb3a4-f37f-4edd-afb1-2190cd1f62fc}
   Get Get: Id {5c8a2ae5-eaad-400d-b638-ec46a75b5ccb}
   Property massMat: Id {c4fbf6a1-1d71-4f80-9bfa-395c19261a6f}
   Get Get: Id {b8079ba8-3835-474b-9d8e-6afd86dc6a9b}
   Property rawJntCurrent: Id {f1221838-7bcd-4d84-b9f8-7dc96a864978}
   Get Get: Id {23a8503d-4e33-47db-b530-039bdd0d530f}
   Property simCartPose: Id {6426ffc4-f74f-4984-ac32-a9f9d8b8c8ca}
   Get Get: Id {a61bb7de-a7ad-4b34-8063-e53c825d0db4}
   Property simJaco: Id {0fa24ffb-bfb3-496c-82de-08842f53e6e4}
   Get Get: Id {35c7dda2-112e-4042-99cd-4eac5d67ff5e}
   Method updateCmds: Id {4f271d3a-4b2b-4f85-986e-f8fdffb5994c}
   Method updateDyna: Id {02de28e3-c8a7-46cf-834a-5bf048b5e039}
   Method updateSimStatus: Id {f15ad7c2-6655-4b50-9555-9aa968e8753f}
   Method updateStatus: Id {21b3fe9a-0eba-4313-bb9a-33b1f0038771} *)
